SUBAPPLICATION Uebung_081 (* Beispiel für E_CTD *)
  (* Standard: 61499-2; Description: Copyright (c) 2023 Meisterschulen am Ostbahnhof This program and the accompanying materials are made available under the terms of the Eclipse Public License 2.0 which is available at https://www.eclipse.org/legal/epl-2.0/ SPDX-License-Identifier: EPL-2.0 Beispiel für E_CTD Aufwärts zählen UAO Curriculum Module 3 - The IEC 61499 Standard, Seite 93 *)
  (* Version 1.0, 2023-10-23, Franz Höpfinger, Meisterschulen am Ostbahnhof *)
  IMPORT logiBUS::io::DI::logiBUS_DI;
  IMPORT logiBUS::io::DI::logiBUS_DI_Events;
  IMPORT logiBUS::io::DQ::logiBUS_DO;
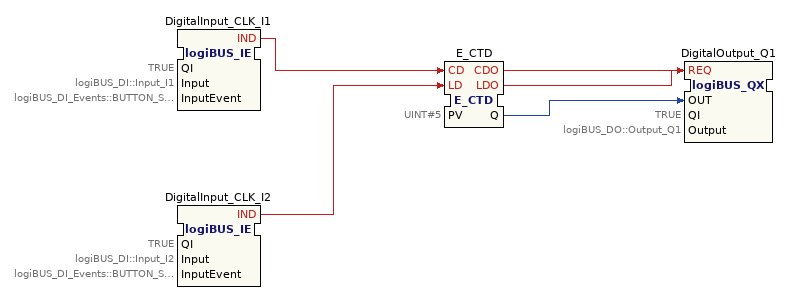
  FBS
    DigitalOutput_Q1 : logiBUS::io::DQ::logiBUS_QX(QI := TRUE, Output := logiBUS_DO::Output_Q1);
    DigitalInput_CLK_I1 : logiBUS::io::DI::logiBUS_IE(QI := TRUE, Input := logiBUS_DI::Input_I1, InputEvent := logiBUS_DI_Events::BUTTON_SINGLE_CLICK);
    E_CTD : iec61499::events::E_CTD(PV := UINT#5);
    DigitalInput_CLK_I2 : logiBUS::io::DI::logiBUS_IE(QI := TRUE, Input := logiBUS_DI::Input_I2, InputEvent := logiBUS_DI_Events::BUTTON_SINGLE_CLICK);
  END_FBS
  EVENT_CONNECTIONS
    DigitalInput_CLK_I1.IND TO E_CTD.CD;
    E_CTD.CDO TO DigitalOutput_Q1.REQ;
    E_CTD.LDO TO DigitalOutput_Q1.REQ;
    DigitalInput_CLK_I2.IND TO E_CTD.LD;
  END_CONNECTIONS
  DATA_CONNECTIONS
    E_CTD.Q TO DigitalOutput_Q1.OUT;
  END_CONNECTIONS
END_SUBAPPLICATION
